SUBAPPLICATION Uebung_020i (* DigitalInput_I1 auf DigitalOutput_Q1; E_PULSE; Impulsformend *)
  (* Standard: 61499-2 *)
  (* Version 1.0, 2023-10-23, franz *)
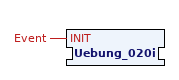
  EVENT_INPUT
    INIT;
  END_EVENT
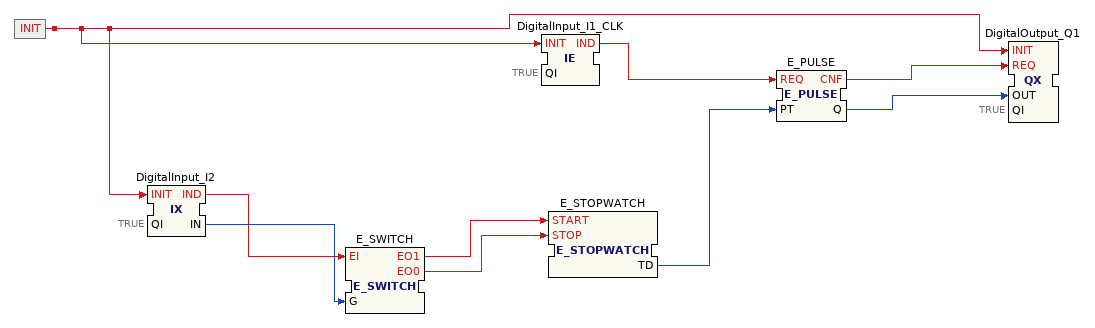
  FBS
    DigitalOutput_Q1 : QX(QI := TRUE);
    E_PULSE : E_PULSE;
    DigitalInput_I1_CLK : IE(QI := TRUE);
    E_STOPWATCH : E_STOPWATCH;
    E_SWITCH : E_SWITCH;
    DigitalInput_I2 : IX(QI := TRUE);
  END_FBS
  EVENT_CONNECTIONS
    INIT TO DigitalOutput_Q1.INIT;
    E_PULSE.CNF TO DigitalOutput_Q1.REQ;
    DigitalInput_I1_CLK.IND TO E_PULSE.REQ;
    INIT TO DigitalInput_I1_CLK.INIT;
    DigitalInput_I2.IND TO E_SWITCH.EI;
    E_SWITCH.EO1 TO E_STOPWATCH.START;
    E_SWITCH.EO0 TO E_STOPWATCH.STOP;
    INIT TO DigitalInput_I2.INIT;
  END_CONNECTIONS
  DATA_CONNECTIONS
    E_PULSE.Q TO DigitalOutput_Q1.OUT;
    E_STOPWATCH.TD TO E_PULSE.PT;
    DigitalInput_I2.IN TO E_SWITCH.G;
  END_CONNECTIONS
END_SUBAPPLICATION
